VISUALIZATION Visualization_Trafficlight_system  // 2x2
END_VISUALIZATION

(* stored: Version 1.1.0.1, ProductVersion 3.1.4024.12
   Visu Visualization_Trafficlight_system: Id {0e9ebbf0-9414-4b60-90fd-9243ae83c1a0} *)
